FUNCTION_BLOCK FB_Drill
VAR_INPUT
	bStart : BOOL;
END_VAR
VAR_OUTPUT
END_VAR
VAR
END_VAR

TRANSITION TRANS_Check:
TRANS_Check := bStart;
END_TRANSITION

END_FUNCTION_BLOCK

(* stored: Version 1.1.0.1, ProductVersion 3.1.4024.16
   POU FB_Drill: Id {0fab13f1-c360-4135-8aab-1eb9236f9c07}, SpecialFunc None
   Transition TRANS_Check: Id {3e98b030-fb01-478e-be50-7cbc290f2709} *)
